FUNCTION_BLOCK FB_FlameCannon
VAR
	_Active : BOOL;
	_Level  : LREAL;
END_VAR

PROPERTY Active : BOOL
GET
Active := This^._Active;
END_GET
END_PROPERTY

PROPERTY Level : LREAL
GET
Level := This^._Level;
END_GET
END_PROPERTY

METHOD Off : BOOL
VAR_INPUT
END_VAR
This^._Active := FALSE;
END_METHOD

METHOD On : BOOL
VAR_INPUT
END_VAR
This^._Active := TRUE;
END_METHOD

METHOD SetLevel : BOOL
VAR_INPUT
	Level  : LREAL;
END_VAR
This^._Level := Level;
END_METHOD

END_FUNCTION_BLOCK

(* stored: Version 1.1.0.1, ProductVersion 3.1.4022.18
   POU FB_FlameCannon: Id {e0c8f848-1784-4d41-b2ed-5a7bf2c4ca4b}, SpecialFunc None
   Property Active: Id {622d1617-e0e5-47d4-8c53-b01331bc5e8f}
   Get Get: Id {18b2bf04-4101-42df-87ce-c6a73e92e684}
   Property Level: Id {873ba544-8cd1-4372-8a10-ed0fef254f41}
   Get Get: Id {b5541769-4efd-45f5-ae2f-b0865110b1b5}
   Method Off: Id {70ce79ff-f68f-4508-bec5-6998f8f5977b}
   Method On: Id {f2e7260b-6b26-4802-a0b4-6bb42e04246f}
   Method SetLevel: Id {a5d325a6-d53c-4e33-9db0-d3ee0d3587aa} *)
